(* PLC project 2b9f17cc-6118-46e7-a7df-88c6d716094c.ecp, WAGO e!COCKPIT e!COCKPIT *)
(* stored: creationDateTime 2017-07-13T16:48:36.5158135, modificationDateTime 2017-07-13T16:45:12.6724614 *)

PROGRAM PLC_PRG
  VAR
    i : INT;
  END_VAR

            i:=i+1;
          
END_PROGRAM
